FUNCTION_BLOCK FB_ModeSelector
VAR_INPUT
	//bControlBox : BOOL;
END_VAR
VAR_OUTPUT
END_VAR
VAR
	fbModeVisualization : FB_ModeVisualization;
	fbModeControlBox : FB_ModeControlBox;
	fbMode : I_Mode := fbModeVisualization;
END_VAR

END_FUNCTION_BLOCK

(* stored: Version 1.1.0.1, ProductVersion 3.1.4024.12
   POU FB_ModeSelector: Id {3399322c-221a-4211-a48b-e9157a0453b6}, SpecialFunc None *)
